% RSLogix 500 project Practise-5.RSS, saved by version 8.30.00.16 %
PROJECT "UNTITLED"    % processor: MicroLogix 1000 %

PROGRAM FILES
  LAD 2 "MAIN_PROG"  8 rungs
  LAD 3 "USER_FAULT"  1 rungs
  LAD 4 "HSC_INT"  1 rungs
  LAD 5 "STI_INT"  1 rungs
  LAD 6, 7, 8, 9, 10, 11, 12, 13, 14, 15, 16: only END

DATA FILES
  O0 OUTPUT  1 elements
  I1 INPUT  2 elements
  S2 STATUS  33 elements
  B3 BINARY  32 elements
  T4 TIMER  40 elements
  C5 COUNTER  32 elements
  R6 CONTROL  16 elements
  N7 INTEGER  105 elements

LADDER 2 "MAIN_PROG"
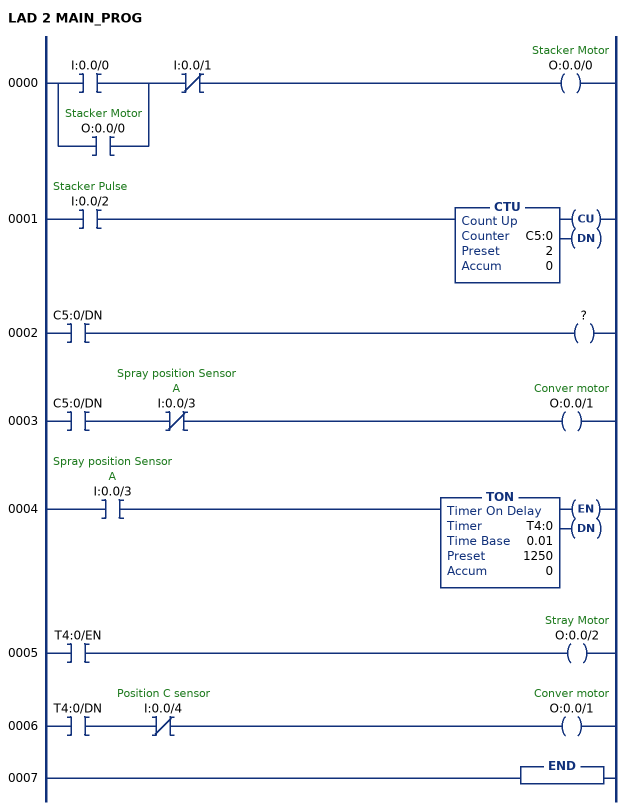
% Rung: 0 %
SOR BST XIC I:0.0/0 NXB XIC O:0.0/0 BND XIO I:0.0/1 OTE O:0.0/0 EOR
%   O:0.0/0  "Stacker Motor" %
% Rung: 1 %  % edit flag set %
SOR XIC I:0.0/2 CTU C5:0 2 0 EOR
%   I:0.0/2  "Stacker Pulse" %
% Rung: 2 %  % edit flag set %
SOR XIC C5:0/DN OTE ? EOR
% Rung: 3 %
SOR XIC C5:0/DN XIO I:0.0/3 OTE O:0.0/1 EOR
%   I:0.0/3  "Spray position Sensor A" %
%   O:0.0/1  "Conver motor" %
% Rung: 4 %
SOR XIC I:0.0/3 TON T4:0 0.01 1250 0 EOR
%   I:0.0/3  "Spray position Sensor A" %
% Rung: 5 %
SOR XIC T4:0/EN OTE O:0.0/2 EOR
%   O:0.0/2  "Stray Motor" %
% Rung: 6 %
SOR XIC T4:0/DN XIO I:0.0/4 OTE O:0.0/1 EOR
%   I:0.0/4  "Position C sensor" %
%   O:0.0/1  "Conver motor" %
% Rung: 7 %
SOR END EOR

DATA TABLE (non-zero values as saved)
DATA T4
% .PRE .ACC %
% T4:0 % 1250 0
DATA C5
% .PRE .ACC %
% C5:0 % 2 0
